{attribute 'qualified_only'}
{attribute 'strict'}
TYPE ST115_PnpVerPushPos_e :
(
	down,
	up,
	_max
);
END_TYPE

(* stored: Version 1.1.0.1, ProductVersion 3.1.4024.6
   DUT ST115_PnpVerPushPos_e: Id {060a9239-b60a-4807-89b3-08d90aafd75e} *)
